// TIA Portal project "Connect_Winform" (V15)

(* hardware
DEVICE "S7-1200 station_1"  S7-1200 Station
   slot 0: "Rack_0"  S7-1200 Rack  Rack  V1.0
   slot 1: "PLC_1"  CPU 1214C DC/DC/Rly  6ES7 214-1HG40-0XB0  V4.2
   slot 2: "DI 16/DQ 16x24VDC_1"  SM 1223 DI16/DQ16 x 24VDC  6ES7 223-1BL30-0XB0  V1.0
*)

// ===== PLC "PLC_1"  CPU 1214C DC/DC/Rly =====

VAR_GLOBAL   // PLC tag table "Input"
   "Man" AT %I0.0 : Bool;
   "Silo1" AT %I0.1 : Bool;
   "Silo2" AT %I0.2 : Bool;
   "Silo3" AT %I0.3 : Bool;
   "Silo4" AT %I0.4 : Bool;
   "Silo5" AT %I0.5 : Bool;
   "Silo6" AT %I0.6 : Bool;
   "Silo7" AT %I0.7 : Bool;
   "Silo8" AT %I8.0 : Bool;
   "Silo9" AT %I8.1 : Bool;
   "Silo10" AT %I8.2 : Bool;
   "Silo11" AT %I8.3 : Bool;
   "Silo12" AT %I8.4 : Bool;
   "Silo13" AT %I8.5 : Bool;
   "Silo14" AT %I8.6 : Bool;
   "Silo15" AT %I8.7 : Bool;
   "Auto" AT %I9.0 : Bool;
   "InSilo" AT %I9.1 : Bool;
   "Mo Can" AT %I9.2 : Bool;
   "Dong Can" AT %I9.3 : Bool;
END_VAR

VAR_GLOBAL   // PLC tag table "Output"
   "Dang Can" AT %Q0.0 : Bool;
   "Silo_1" AT %Q0.1 : Bool;
   "Silo_2" AT %Q0.2 : Bool;
   "Silo_3" AT %Q0.3 : Bool;
   "Silo_4" AT %Q0.4 : Bool;
   "Silo_5" AT %Q0.5 : Bool;
   "Silo_6" AT %Q9.1 : Bool;
   "Silo_7" AT %Q9.2 : Bool;
   "Silo_8" AT %Q8.0 : Bool;
   "Silo_9" AT %Q8.1 : Bool;
   "Silo_10" AT %Q8.2 : Bool;
   "Silo_11" AT %Q8.3 : Bool;
   "Silo_12" AT %Q8.4 : Bool;
   "Silo_13" AT %Q8.5 : Bool;
   "Silo_14" AT %Q8.6 : Bool;
   "Silo_15" AT %Q8.7 : Bool;
   "Ngung Can" AT %Q9.0 : Bool;
   "Silo_16" AT %Q9.3 : Bool;
END_VAR

VAR_GLOBAL   // PLC tag table "Bien_Trung_Gian"
   "Bang_Tay" AT %M0.0 : Bool;
   "Sl1" AT %M0.1 : Bool;
   "Sl2" AT %M0.2 : Bool;
   "Sl3" AT %M0.3 : Bool;
   "Sl4" AT %M0.4 : Bool;
   "Sl5" AT %M0.5 : Bool;
   "Sl6" AT %M0.6 : Bool;
   "Sl7" AT %M0.7 : Bool;
   "Sl8" AT %M1.0 : Bool;
   "Sl9" AT %M1.1 : Bool;
   "Sl10" AT %M1.2 : Bool;
   "Sl11" AT %M1.3 : Bool;
   "Sl12" AT %M1.4 : Bool;
   "Sl13" AT %M1.5 : Bool;
   "Sl14" AT %M1.6 : Bool;
   "Sl15" AT %M1.7 : Bool;
   "Tu_Dong" AT %M2.0 : Bool;
   "Cho_Phep_Can1" AT %M2.1 : Bool;
   "Cho_Xa_Can" AT %M2.2 : Bool;
   "Sl16" AT %M2.3 : Bool;
   "Cho_Phep_Can2" AT %M2.4 : Bool;
   "Cho_Phep_Can3" AT %M2.5 : Bool;
END_VAR

DATA_BLOCK "DB_Winform"   // DB1
{ S7_Optimized_Access := 'FALSE' }
VERSION : 0.1
   VAR
      sn : Bool;
      Den2 : Bool;
      Den3 : Bool;
      Den4 : Bool;
      Den5 : Bool;
      Den6 : Bool;
      Den7 : Bool;
      Den8 : Bool;
      Den9 : Bool;
      Den10 : Bool;
      Den11 : Bool;
      Den12 : Bool;
      Den13 : Bool;
      Den14 : Bool;
      Den15 : Bool;
      Den16 : Bool;
      Den_CPC1 : Bool;
      Den_CPC2 : Bool;
      Den_CPC3 : Bool;
      end : Byte;
   END_VAR
BEGIN
END_DATA_BLOCK

DATA_BLOCK "FB1_Silo1"   // DB2
{ S7_Optimized_Access := 'TRUE' }
VERSION : 0.1
// stored: InstanceOfName FB1
"FB1"
BEGIN
END_DATA_BLOCK

DATA_BLOCK "FB1_Silo2"   // DB3
{ S7_Optimized_Access := 'TRUE' }
VERSION : 0.1
// stored: InstanceOfName FB1
"FB1"
BEGIN
END_DATA_BLOCK

DATA_BLOCK "FB1_Silo3"   // DB4
{ S7_Optimized_Access := 'TRUE' }
VERSION : 0.1
// stored: InstanceOfName FB1
"FB1"
BEGIN
END_DATA_BLOCK

DATA_BLOCK "FB1_Silo4"   // DB5
{ S7_Optimized_Access := 'TRUE' }
VERSION : 0.1
// stored: InstanceOfName FB1
"FB1"
BEGIN
END_DATA_BLOCK

DATA_BLOCK "FB1_Silo5"   // DB6
{ S7_Optimized_Access := 'TRUE' }
VERSION : 0.1
// stored: InstanceOfName FB1
"FB1"
BEGIN
END_DATA_BLOCK

DATA_BLOCK "FB1_Silo6"   // DB7
{ S7_Optimized_Access := 'TRUE' }
VERSION : 0.1
// stored: InstanceOfName FB1
"FB1"
BEGIN
END_DATA_BLOCK

DATA_BLOCK "FB1_Silo7"   // DB8
{ S7_Optimized_Access := 'TRUE' }
VERSION : 0.1
// stored: InstanceOfName FB1
"FB1"
BEGIN
END_DATA_BLOCK

DATA_BLOCK "FB1_Silo8"   // DB9
{ S7_Optimized_Access := 'TRUE' }
VERSION : 0.1
// stored: InstanceOfName FB1
"FB1"
BEGIN
END_DATA_BLOCK

DATA_BLOCK "FB1_Silo9"   // DB10
{ S7_Optimized_Access := 'TRUE' }
VERSION : 0.1
// stored: InstanceOfName FB1
"FB1"
BEGIN
END_DATA_BLOCK

DATA_BLOCK "FB1_Silo10"   // DB11
{ S7_Optimized_Access := 'TRUE' }
VERSION : 0.1
// stored: InstanceOfName FB1
"FB1"
BEGIN
END_DATA_BLOCK

DATA_BLOCK "FB1_Silo11"   // DB12
{ S7_Optimized_Access := 'TRUE' }
VERSION : 0.1
// stored: InstanceOfName FB1
"FB1"
BEGIN
END_DATA_BLOCK

DATA_BLOCK "FB1_Silo12"   // DB13
{ S7_Optimized_Access := 'TRUE' }
VERSION : 0.1
// stored: InstanceOfName FB1
"FB1"
BEGIN
END_DATA_BLOCK

DATA_BLOCK "FB1_Silo13"   // DB14
{ S7_Optimized_Access := 'TRUE' }
VERSION : 0.1
// stored: InstanceOfName FB1
"FB1"
BEGIN
END_DATA_BLOCK

DATA_BLOCK "FB1_Silo14"   // DB15
{ S7_Optimized_Access := 'TRUE' }
VERSION : 0.1
// stored: InstanceOfName FB1
"FB1"
BEGIN
END_DATA_BLOCK

DATA_BLOCK "FB1_Silo15"   // DB16
{ S7_Optimized_Access := 'TRUE' }
VERSION : 0.1
// stored: InstanceOfName FB1
"FB1"
BEGIN
END_DATA_BLOCK

DATA_BLOCK "FB1_Silo16"   // DB17
{ S7_Optimized_Access := 'TRUE' }
VERSION : 0.1
// stored: InstanceOfName FB1
"FB1"
BEGIN
END_DATA_BLOCK

FUNCTION_BLOCK "FB1"   // FB1, LAD
{ S7_Optimized_Access := 'TRUE' }
VERSION : 0.1
   VAR_INPUT
      Silo : Bool;
      "Silo+1" : Bool;
      "Silo+2" : Bool;
      "Silo+3" : Bool;
      "Silo+4" : Bool;
      "Silo+5" : Bool;
      "Silo+6" : Bool;
      "Silo+7" : Bool;
      "Silo+8" : Bool;
      "Silo+9" : Bool;
      "Silo+10" : Bool;
      "Silo+11" : Bool;
      "Silo+12" : Bool;
      "Silo+13" : Bool;
      "Silo+14" : Bool;
      "Silo+15" : Bool;
      In_Silo : Bool;
      Cho_Phep_Can : Bool;
      Nhan_Giu : Bool;
   END_VAR
   VAR_OUTPUT
      Silo_On : Bool;
   END_VAR
BEGIN

REGION Network 1
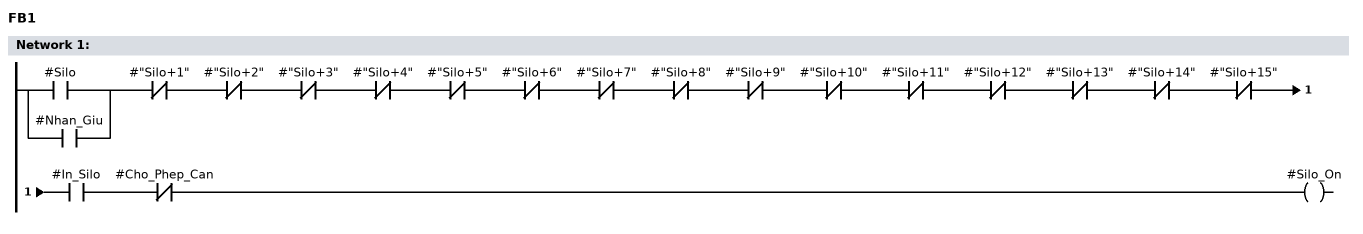
   RUNG wire#powerrail
      Contact( #Silo )
      wire#w1
      I_Contact( #"Silo+1" )
      I_Contact( #"Silo+2" )
      I_Contact( #"Silo+3" )
      I_Contact( #"Silo+4" )
      I_Contact( #"Silo+5" )
      I_Contact( #"Silo+6" )
      I_Contact( #"Silo+7" )
      I_Contact( #"Silo+8" )
      I_Contact( #"Silo+9" )
      I_Contact( #"Silo+10" )
      I_Contact( #"Silo+11" )
      I_Contact( #"Silo+12" )
      I_Contact( #"Silo+13" )
      I_Contact( #"Silo+14" )
      I_Contact( #"Silo+15" )
      Contact( #In_Silo )
      I_Contact( #Cho_Phep_Can )
      Coil( #Silo_On )
   END_RUNG
   RUNG wire#powerrail
      Contact( #Nhan_Giu )
   END_RUNG wire#w1
   // the same network as SCL:
   #Silo_On := (#Silo OR #Nhan_Giu) AND NOT #"Silo+1" AND NOT #"Silo+2" AND NOT #"Silo+3" AND NOT #"Silo+4" AND NOT #"Silo+5" AND NOT #"Silo+6" AND NOT #"Silo+7" AND NOT #"Silo+8" AND NOT #"Silo+9" AND NOT #"Silo+10" AND NOT #"Silo+11" AND NOT #"Silo+12" AND NOT #"Silo+13" AND NOT #"Silo+14" AND NOT #"Silo+15" AND #In_Silo AND NOT #Cho_Phep_Can;
END_REGION
END_FUNCTION_BLOCK

ORGANIZATION_BLOCK "Can"   // OB1, LAD, ProgramCycle
TITLE = "Main Program Sweep (Cycle)"
{ S7_Optimized_Access := 'TRUE' }
VERSION : 0.1
   VAR_INPUT
      Initial_Call : Bool;   // Initial call of this OB
      Remanence : Bool;   // =True, if remanent data are available
   END_VAR
BEGIN

REGION Network 1
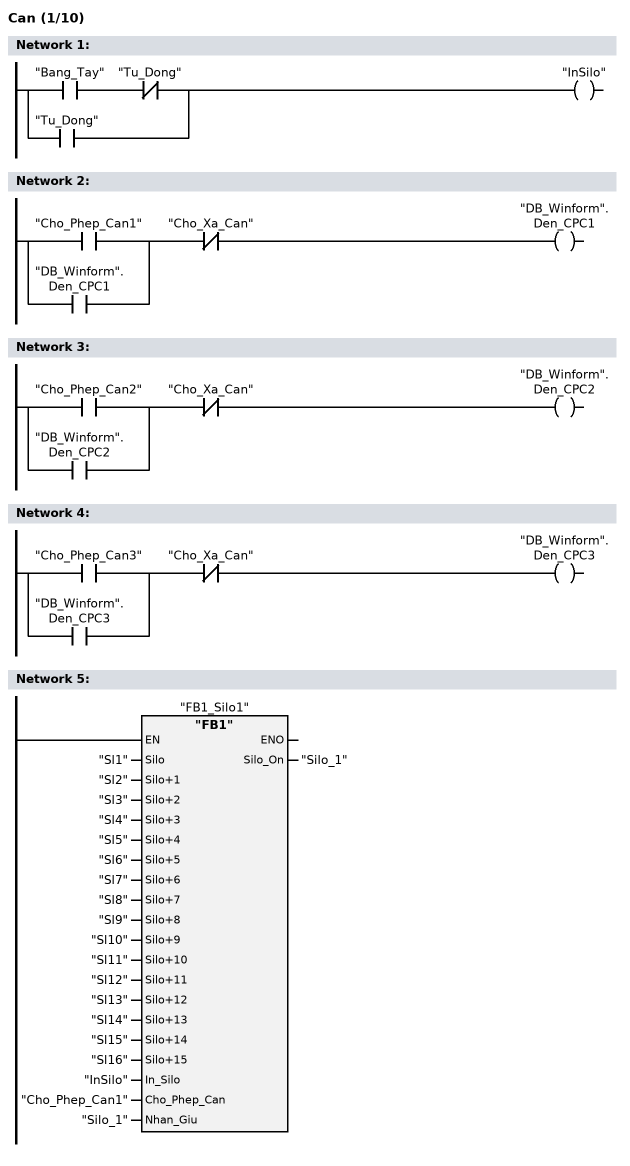
   RUNG wire#powerrail
      Contact( "Bang_Tay" )
      I_Contact( "Tu_Dong" )
      wire#w1
      Coil( "InSilo" )
   END_RUNG
   RUNG wire#powerrail
      Contact( "Tu_Dong" )
   END_RUNG wire#w1
   // the same network as SCL:
   "InSilo" := ("Bang_Tay" AND NOT "Tu_Dong") OR "Tu_Dong";
END_REGION

REGION Network 2
   RUNG wire#powerrail
      Contact( "Cho_Phep_Can1" )
      wire#w1
      I_Contact( "Cho_Xa_Can" )
      Coil( "DB_Winform".Den_CPC1 )
   END_RUNG
   RUNG wire#powerrail
      Contact( "DB_Winform".Den_CPC1 )
   END_RUNG wire#w1
   // the same network as SCL:
   "DB_Winform".Den_CPC1 := ("Cho_Phep_Can1" OR "DB_Winform".Den_CPC1) AND NOT "Cho_Xa_Can";
END_REGION

REGION Network 3
   RUNG wire#powerrail
      Contact( "Cho_Phep_Can2" )
      wire#w1
      I_Contact( "Cho_Xa_Can" )
      Coil( "DB_Winform".Den_CPC2 )
   END_RUNG
   RUNG wire#powerrail
      Contact( "DB_Winform".Den_CPC2 )
   END_RUNG wire#w1
   // the same network as SCL:
   "DB_Winform".Den_CPC2 := ("Cho_Phep_Can2" OR "DB_Winform".Den_CPC2) AND NOT "Cho_Xa_Can";
END_REGION

REGION Network 4
   RUNG wire#powerrail
      Contact( "Cho_Phep_Can3" )
      wire#w1
      I_Contact( "Cho_Xa_Can" )
      Coil( "DB_Winform".Den_CPC3 )
   END_RUNG
   RUNG wire#powerrail
      Contact( "DB_Winform".Den_CPC3 )
   END_RUNG wire#w1
   // the same network as SCL:
   "DB_Winform".Den_CPC3 := ("Cho_Phep_Can3" OR "DB_Winform".Den_CPC3) AND NOT "Cho_Xa_Can";
END_REGION

REGION Network 5
   RUNG wire#powerrail
      "FB1_Silo1"(Silo := "Sl1", "Silo+1" := "Sl2", "Silo+2" := "Sl3", "Silo+3" := "Sl4", "Silo+4" := "Sl5", "Silo+5" := "Sl6", "Silo+6" := "Sl7", "Silo+7" := "Sl8", "Silo+8" := "Sl9", "Silo+9" := "Sl10", "Silo+10" := "Sl11", "Silo+11" := "Sl12", "Silo+12" := "Sl13", "Silo+13" := "Sl14", "Silo+14" := "Sl15", "Silo+15" := "Sl16", In_Silo := "InSilo", Cho_Phep_Can := "Cho_Phep_Can1", Nhan_Giu := "Silo_1", Silo_On => "Silo_1")
   END_RUNG
   // the same network as SCL:
   "FB1_Silo1"(Silo := "Sl1",   // "FB1"
               "Silo+1" := "Sl2",
               "Silo+2" := "Sl3",
               "Silo+3" := "Sl4",
               "Silo+4" := "Sl5",
               "Silo+5" := "Sl6",
               "Silo+6" := "Sl7",
               "Silo+7" := "Sl8",
               "Silo+8" := "Sl9",
               "Silo+9" := "Sl10",
               "Silo+10" := "Sl11",
               "Silo+11" := "Sl12",
               "Silo+12" := "Sl13",
               "Silo+13" := "Sl14",
               "Silo+14" := "Sl15",
               "Silo+15" := "Sl16",
               In_Silo := "InSilo",
               Cho_Phep_Can := "Cho_Phep_Can1",
               Nhan_Giu := "Silo_1",
               Silo_On => "Silo_1");
END_REGION

REGION Network 6
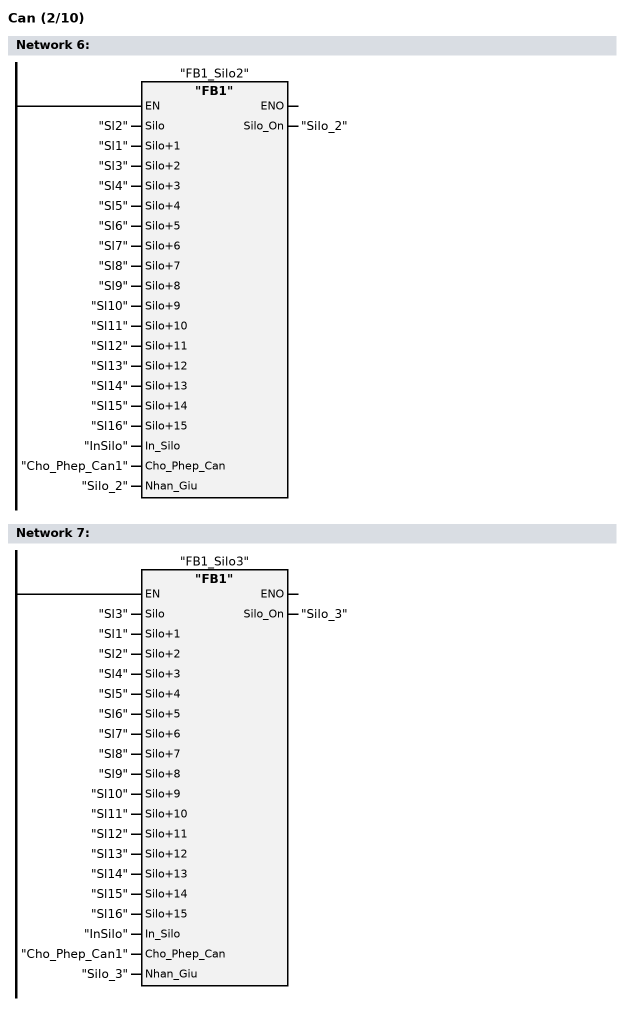
   RUNG wire#powerrail
      "FB1_Silo2"(Silo := "Sl2", "Silo+1" := "Sl1", "Silo+2" := "Sl3", "Silo+3" := "Sl4", "Silo+4" := "Sl5", "Silo+5" := "Sl6", "Silo+6" := "Sl7", "Silo+7" := "Sl8", "Silo+8" := "Sl9", "Silo+9" := "Sl10", "Silo+10" := "Sl11", "Silo+11" := "Sl12", "Silo+12" := "Sl13", "Silo+13" := "Sl14", "Silo+14" := "Sl15", "Silo+15" := "Sl16", In_Silo := "InSilo", Cho_Phep_Can := "Cho_Phep_Can1", Nhan_Giu := "Silo_2", Silo_On => "Silo_2")
   END_RUNG
   // the same network as SCL:
   "FB1_Silo2"(Silo := "Sl2",   // "FB1"
               "Silo+1" := "Sl1",
               "Silo+2" := "Sl3",
               "Silo+3" := "Sl4",
               "Silo+4" := "Sl5",
               "Silo+5" := "Sl6",
               "Silo+6" := "Sl7",
               "Silo+7" := "Sl8",
               "Silo+8" := "Sl9",
               "Silo+9" := "Sl10",
               "Silo+10" := "Sl11",
               "Silo+11" := "Sl12",
               "Silo+12" := "Sl13",
               "Silo+13" := "Sl14",
               "Silo+14" := "Sl15",
               "Silo+15" := "Sl16",
               In_Silo := "InSilo",
               Cho_Phep_Can := "Cho_Phep_Can1",
               Nhan_Giu := "Silo_2",
               Silo_On => "Silo_2");
END_REGION

REGION Network 7
   RUNG wire#powerrail
      "FB1_Silo3"(Silo := "Sl3", "Silo+1" := "Sl1", "Silo+2" := "Sl2", "Silo+3" := "Sl4", "Silo+4" := "Sl5", "Silo+5" := "Sl6", "Silo+6" := "Sl7", "Silo+7" := "Sl8", "Silo+8" := "Sl9", "Silo+9" := "Sl10", "Silo+10" := "Sl11", "Silo+11" := "Sl12", "Silo+12" := "Sl13", "Silo+13" := "Sl14", "Silo+14" := "Sl15", "Silo+15" := "Sl16", In_Silo := "InSilo", Cho_Phep_Can := "Cho_Phep_Can1", Nhan_Giu := "Silo_3", Silo_On => "Silo_3")
   END_RUNG
   // the same network as SCL:
   "FB1_Silo3"(Silo := "Sl3",   // "FB1"
               "Silo+1" := "Sl1",
               "Silo+2" := "Sl2",
               "Silo+3" := "Sl4",
               "Silo+4" := "Sl5",
               "Silo+5" := "Sl6",
               "Silo+6" := "Sl7",
               "Silo+7" := "Sl8",
               "Silo+8" := "Sl9",
               "Silo+9" := "Sl10",
               "Silo+10" := "Sl11",
               "Silo+11" := "Sl12",
               "Silo+12" := "Sl13",
               "Silo+13" := "Sl14",
               "Silo+14" := "Sl15",
               "Silo+15" := "Sl16",
               In_Silo := "InSilo",
               Cho_Phep_Can := "Cho_Phep_Can1",
               Nhan_Giu := "Silo_3",
               Silo_On => "Silo_3");
END_REGION

REGION Network 8
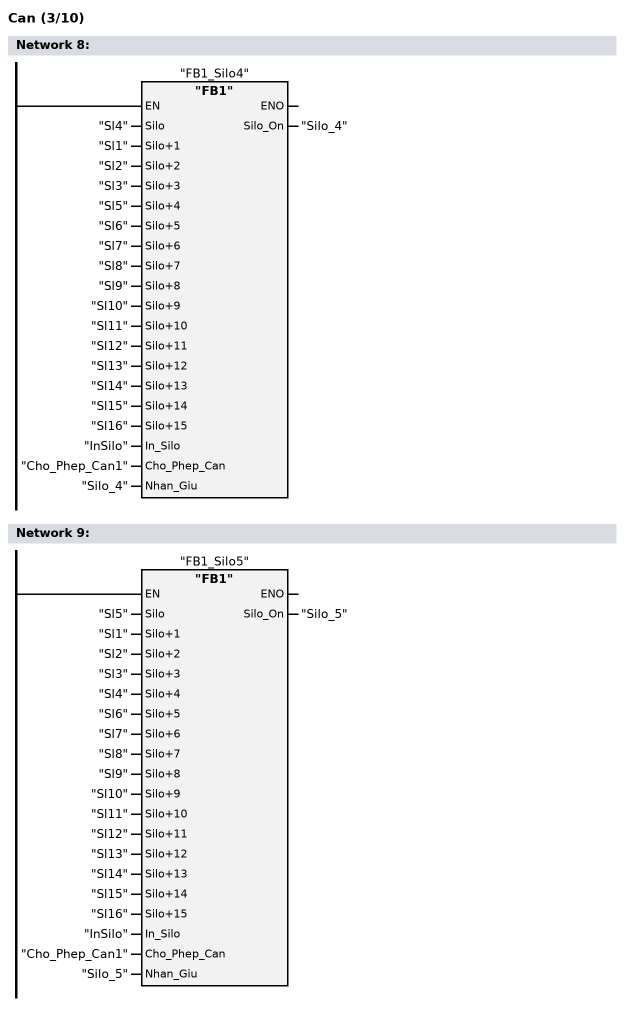
   RUNG wire#powerrail
      "FB1_Silo4"(Silo := "Sl4", "Silo+1" := "Sl1", "Silo+2" := "Sl2", "Silo+3" := "Sl3", "Silo+4" := "Sl5", "Silo+5" := "Sl6", "Silo+6" := "Sl7", "Silo+7" := "Sl8", "Silo+8" := "Sl9", "Silo+9" := "Sl10", "Silo+10" := "Sl11", "Silo+11" := "Sl12", "Silo+12" := "Sl13", "Silo+13" := "Sl14", "Silo+14" := "Sl15", "Silo+15" := "Sl16", In_Silo := "InSilo", Cho_Phep_Can := "Cho_Phep_Can1", Nhan_Giu := "Silo_4", Silo_On => "Silo_4")
   END_RUNG
   // the same network as SCL:
   "FB1_Silo4"(Silo := "Sl4",   // "FB1"
               "Silo+1" := "Sl1",
               "Silo+2" := "Sl2",
               "Silo+3" := "Sl3",
               "Silo+4" := "Sl5",
               "Silo+5" := "Sl6",
               "Silo+6" := "Sl7",
               "Silo+7" := "Sl8",
               "Silo+8" := "Sl9",
               "Silo+9" := "Sl10",
               "Silo+10" := "Sl11",
               "Silo+11" := "Sl12",
               "Silo+12" := "Sl13",
               "Silo+13" := "Sl14",
               "Silo+14" := "Sl15",
               "Silo+15" := "Sl16",
               In_Silo := "InSilo",
               Cho_Phep_Can := "Cho_Phep_Can1",
               Nhan_Giu := "Silo_4",
               Silo_On => "Silo_4");
END_REGION

REGION Network 9
   RUNG wire#powerrail
      "FB1_Silo5"(Silo := "Sl5", "Silo+1" := "Sl1", "Silo+2" := "Sl2", "Silo+3" := "Sl3", "Silo+4" := "Sl4", "Silo+5" := "Sl6", "Silo+6" := "Sl7", "Silo+7" := "Sl8", "Silo+8" := "Sl9", "Silo+9" := "Sl10", "Silo+10" := "Sl11", "Silo+11" := "Sl12", "Silo+12" := "Sl13", "Silo+13" := "Sl14", "Silo+14" := "Sl15", "Silo+15" := "Sl16", In_Silo := "InSilo", Cho_Phep_Can := "Cho_Phep_Can1", Nhan_Giu := "Silo_5", Silo_On => "Silo_5")
   END_RUNG
   // the same network as SCL:
   "FB1_Silo5"(Silo := "Sl5",   // "FB1"
               "Silo+1" := "Sl1",
               "Silo+2" := "Sl2",
               "Silo+3" := "Sl3",
               "Silo+4" := "Sl4",
               "Silo+5" := "Sl6",
               "Silo+6" := "Sl7",
               "Silo+7" := "Sl8",
               "Silo+8" := "Sl9",
               "Silo+9" := "Sl10",
               "Silo+10" := "Sl11",
               "Silo+11" := "Sl12",
               "Silo+12" := "Sl13",
               "Silo+13" := "Sl14",
               "Silo+14" := "Sl15",
               "Silo+15" := "Sl16",
               In_Silo := "InSilo",
               Cho_Phep_Can := "Cho_Phep_Can1",
               Nhan_Giu := "Silo_5",
               Silo_On => "Silo_5");
END_REGION

REGION Network 10
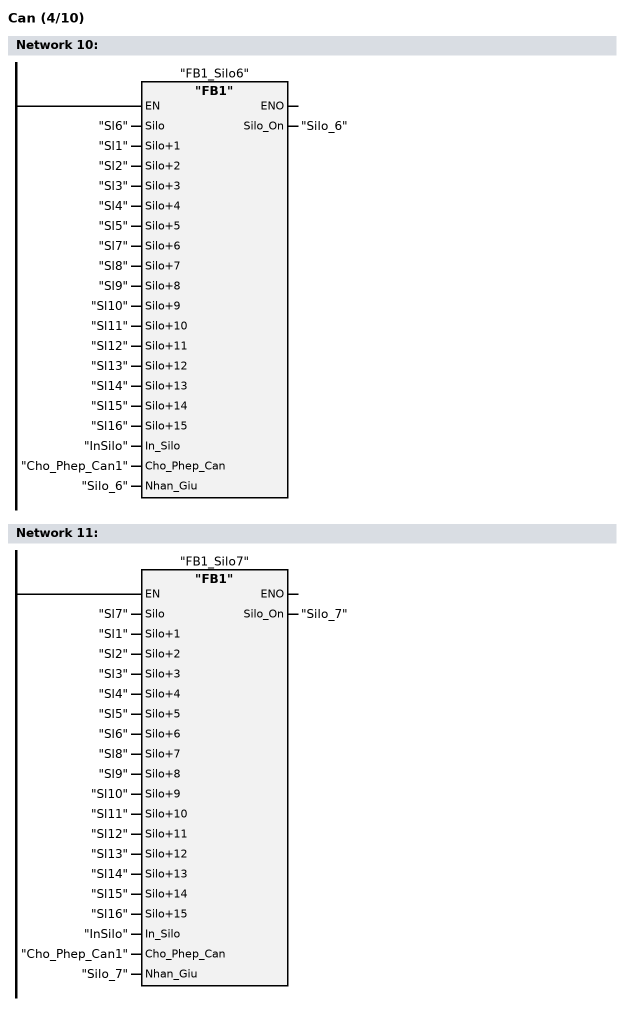
   RUNG wire#powerrail
      "FB1_Silo6"(Silo := "Sl6", "Silo+1" := "Sl1", "Silo+2" := "Sl2", "Silo+3" := "Sl3", "Silo+4" := "Sl4", "Silo+5" := "Sl5", "Silo+6" := "Sl7", "Silo+7" := "Sl8", "Silo+8" := "Sl9", "Silo+9" := "Sl10", "Silo+10" := "Sl11", "Silo+11" := "Sl12", "Silo+12" := "Sl13", "Silo+13" := "Sl14", "Silo+14" := "Sl15", "Silo+15" := "Sl16", In_Silo := "InSilo", Cho_Phep_Can := "Cho_Phep_Can1", Nhan_Giu := "Silo_6", Silo_On => "Silo_6")
   END_RUNG
   // the same network as SCL:
   "FB1_Silo6"(Silo := "Sl6",   // "FB1"
               "Silo+1" := "Sl1",
               "Silo+2" := "Sl2",
               "Silo+3" := "Sl3",
               "Silo+4" := "Sl4",
               "Silo+5" := "Sl5",
               "Silo+6" := "Sl7",
               "Silo+7" := "Sl8",
               "Silo+8" := "Sl9",
               "Silo+9" := "Sl10",
               "Silo+10" := "Sl11",
               "Silo+11" := "Sl12",
               "Silo+12" := "Sl13",
               "Silo+13" := "Sl14",
               "Silo+14" := "Sl15",
               "Silo+15" := "Sl16",
               In_Silo := "InSilo",
               Cho_Phep_Can := "Cho_Phep_Can1",
               Nhan_Giu := "Silo_6",
               Silo_On => "Silo_6");
END_REGION

REGION Network 11
   RUNG wire#powerrail
      "FB1_Silo7"(Silo := "Sl7", "Silo+1" := "Sl1", "Silo+2" := "Sl2", "Silo+3" := "Sl3", "Silo+4" := "Sl4", "Silo+5" := "Sl5", "Silo+6" := "Sl6", "Silo+7" := "Sl8", "Silo+8" := "Sl9", "Silo+9" := "Sl10", "Silo+10" := "Sl11", "Silo+11" := "Sl12", "Silo+12" := "Sl13", "Silo+13" := "Sl14", "Silo+14" := "Sl15", "Silo+15" := "Sl16", In_Silo := "InSilo", Cho_Phep_Can := "Cho_Phep_Can1", Nhan_Giu := "Silo_7", Silo_On => "Silo_7")
   END_RUNG
   // the same network as SCL:
   "FB1_Silo7"(Silo := "Sl7",   // "FB1"
               "Silo+1" := "Sl1",
               "Silo+2" := "Sl2",
               "Silo+3" := "Sl3",
               "Silo+4" := "Sl4",
               "Silo+5" := "Sl5",
               "Silo+6" := "Sl6",
               "Silo+7" := "Sl8",
               "Silo+8" := "Sl9",
               "Silo+9" := "Sl10",
               "Silo+10" := "Sl11",
               "Silo+11" := "Sl12",
               "Silo+12" := "Sl13",
               "Silo+13" := "Sl14",
               "Silo+14" := "Sl15",
               "Silo+15" := "Sl16",
               In_Silo := "InSilo",
               Cho_Phep_Can := "Cho_Phep_Can1",
               Nhan_Giu := "Silo_7",
               Silo_On => "Silo_7");
END_REGION

REGION Network 12
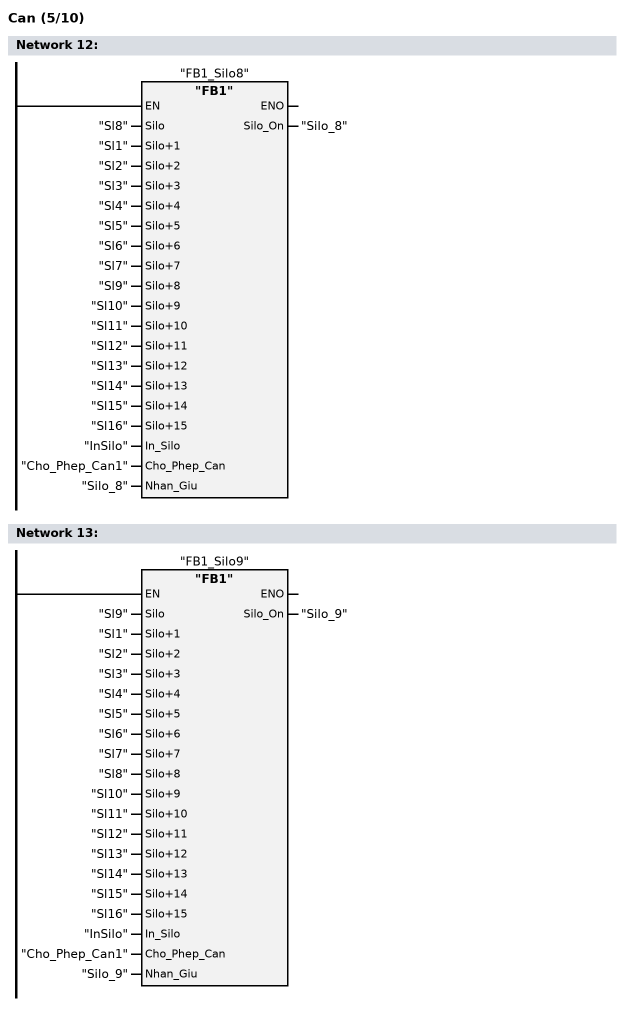
   RUNG wire#powerrail
      "FB1_Silo8"(Silo := "Sl8", "Silo+1" := "Sl1", "Silo+2" := "Sl2", "Silo+3" := "Sl3", "Silo+4" := "Sl4", "Silo+5" := "Sl5", "Silo+6" := "Sl6", "Silo+7" := "Sl7", "Silo+8" := "Sl9", "Silo+9" := "Sl10", "Silo+10" := "Sl11", "Silo+11" := "Sl12", "Silo+12" := "Sl13", "Silo+13" := "Sl14", "Silo+14" := "Sl15", "Silo+15" := "Sl16", In_Silo := "InSilo", Cho_Phep_Can := "Cho_Phep_Can1", Nhan_Giu := "Silo_8", Silo_On => "Silo_8")
   END_RUNG
   // the same network as SCL:
   "FB1_Silo8"(Silo := "Sl8",   // "FB1"
               "Silo+1" := "Sl1",
               "Silo+2" := "Sl2",
               "Silo+3" := "Sl3",
               "Silo+4" := "Sl4",
               "Silo+5" := "Sl5",
               "Silo+6" := "Sl6",
               "Silo+7" := "Sl7",
               "Silo+8" := "Sl9",
               "Silo+9" := "Sl10",
               "Silo+10" := "Sl11",
               "Silo+11" := "Sl12",
               "Silo+12" := "Sl13",
               "Silo+13" := "Sl14",
               "Silo+14" := "Sl15",
               "Silo+15" := "Sl16",
               In_Silo := "InSilo",
               Cho_Phep_Can := "Cho_Phep_Can1",
               Nhan_Giu := "Silo_8",
               Silo_On => "Silo_8");
END_REGION

REGION Network 13
   RUNG wire#powerrail
      "FB1_Silo9"(Silo := "Sl9", "Silo+1" := "Sl1", "Silo+2" := "Sl2", "Silo+3" := "Sl3", "Silo+4" := "Sl4", "Silo+5" := "Sl5", "Silo+6" := "Sl6", "Silo+7" := "Sl7", "Silo+8" := "Sl8", "Silo+9" := "Sl10", "Silo+10" := "Sl11", "Silo+11" := "Sl12", "Silo+12" := "Sl13", "Silo+13" := "Sl14", "Silo+14" := "Sl15", "Silo+15" := "Sl16", In_Silo := "InSilo", Cho_Phep_Can := "Cho_Phep_Can1", Nhan_Giu := "Silo_9", Silo_On => "Silo_9")
   END_RUNG
   // the same network as SCL:
   "FB1_Silo9"(Silo := "Sl9",   // "FB1"
               "Silo+1" := "Sl1",
               "Silo+2" := "Sl2",
               "Silo+3" := "Sl3",
               "Silo+4" := "Sl4",
               "Silo+5" := "Sl5",
               "Silo+6" := "Sl6",
               "Silo+7" := "Sl7",
               "Silo+8" := "Sl8",
               "Silo+9" := "Sl10",
               "Silo+10" := "Sl11",
               "Silo+11" := "Sl12",
               "Silo+12" := "Sl13",
               "Silo+13" := "Sl14",
               "Silo+14" := "Sl15",
               "Silo+15" := "Sl16",
               In_Silo := "InSilo",
               Cho_Phep_Can := "Cho_Phep_Can1",
               Nhan_Giu := "Silo_9",
               Silo_On => "Silo_9");
END_REGION

REGION Network 14
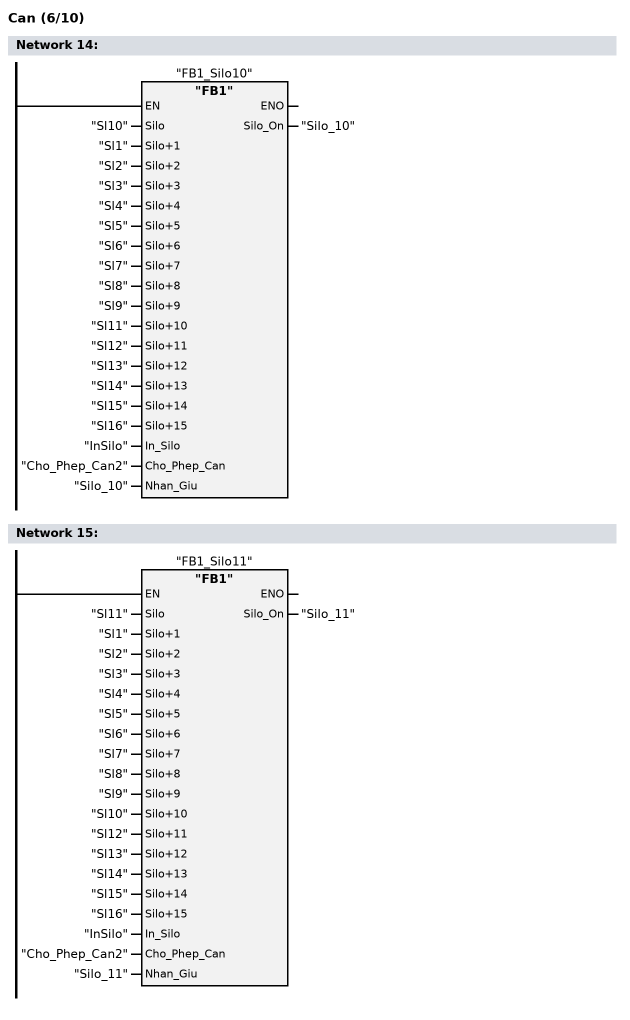
   RUNG wire#powerrail
      "FB1_Silo10"(Silo := "Sl10", "Silo+1" := "Sl1", "Silo+2" := "Sl2", "Silo+3" := "Sl3", "Silo+4" := "Sl4", "Silo+5" := "Sl5", "Silo+6" := "Sl6", "Silo+7" := "Sl7", "Silo+8" := "Sl8", "Silo+9" := "Sl9", "Silo+10" := "Sl11", "Silo+11" := "Sl12", "Silo+12" := "Sl13", "Silo+13" := "Sl14", "Silo+14" := "Sl15", "Silo+15" := "Sl16", In_Silo := "InSilo", Cho_Phep_Can := "Cho_Phep_Can2", Nhan_Giu := "Silo_10", Silo_On => "Silo_10")
   END_RUNG
   // the same network as SCL:
   "FB1_Silo10"(Silo := "Sl10",   // "FB1"
                "Silo+1" := "Sl1",
                "Silo+2" := "Sl2",
                "Silo+3" := "Sl3",
                "Silo+4" := "Sl4",
                "Silo+5" := "Sl5",
                "Silo+6" := "Sl6",
                "Silo+7" := "Sl7",
                "Silo+8" := "Sl8",
                "Silo+9" := "Sl9",
                "Silo+10" := "Sl11",
                "Silo+11" := "Sl12",
                "Silo+12" := "Sl13",
                "Silo+13" := "Sl14",
                "Silo+14" := "Sl15",
                "Silo+15" := "Sl16",
                In_Silo := "InSilo",
                Cho_Phep_Can := "Cho_Phep_Can2",
                Nhan_Giu := "Silo_10",
                Silo_On => "Silo_10");
END_REGION

REGION Network 15
   RUNG wire#powerrail
      "FB1_Silo11"(Silo := "Sl11", "Silo+1" := "Sl1", "Silo+2" := "Sl2", "Silo+3" := "Sl3", "Silo+4" := "Sl4", "Silo+5" := "Sl5", "Silo+6" := "Sl6", "Silo+7" := "Sl7", "Silo+8" := "Sl8", "Silo+9" := "Sl9", "Silo+10" := "Sl10", "Silo+11" := "Sl12", "Silo+12" := "Sl13", "Silo+13" := "Sl14", "Silo+14" := "Sl15", "Silo+15" := "Sl16", In_Silo := "InSilo", Cho_Phep_Can := "Cho_Phep_Can2", Nhan_Giu := "Silo_11", Silo_On => "Silo_11")
   END_RUNG
   // the same network as SCL:
   "FB1_Silo11"(Silo := "Sl11",   // "FB1"
                "Silo+1" := "Sl1",
                "Silo+2" := "Sl2",
                "Silo+3" := "Sl3",
                "Silo+4" := "Sl4",
                "Silo+5" := "Sl5",
                "Silo+6" := "Sl6",
                "Silo+7" := "Sl7",
                "Silo+8" := "Sl8",
                "Silo+9" := "Sl9",
                "Silo+10" := "Sl10",
                "Silo+11" := "Sl12",
                "Silo+12" := "Sl13",
                "Silo+13" := "Sl14",
                "Silo+14" := "Sl15",
                "Silo+15" := "Sl16",
                In_Silo := "InSilo",
                Cho_Phep_Can := "Cho_Phep_Can2",
                Nhan_Giu := "Silo_11",
                Silo_On => "Silo_11");
END_REGION

REGION Network 16
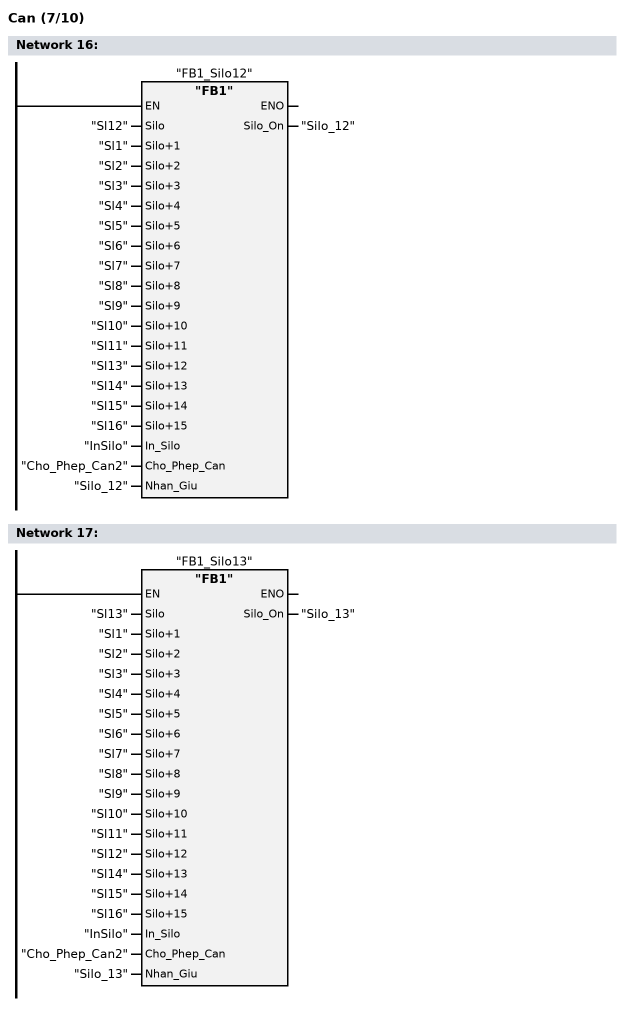
   RUNG wire#powerrail
      "FB1_Silo12"(Silo := "Sl12", "Silo+1" := "Sl1", "Silo+2" := "Sl2", "Silo+3" := "Sl3", "Silo+4" := "Sl4", "Silo+5" := "Sl5", "Silo+6" := "Sl6", "Silo+7" := "Sl7", "Silo+8" := "Sl8", "Silo+9" := "Sl9", "Silo+10" := "Sl10", "Silo+11" := "Sl11", "Silo+12" := "Sl13", "Silo+13" := "Sl14", "Silo+14" := "Sl15", "Silo+15" := "Sl16", In_Silo := "InSilo", Cho_Phep_Can := "Cho_Phep_Can2", Nhan_Giu := "Silo_12", Silo_On => "Silo_12")
   END_RUNG
   // the same network as SCL:
   "FB1_Silo12"(Silo := "Sl12",   // "FB1"
                "Silo+1" := "Sl1",
                "Silo+2" := "Sl2",
                "Silo+3" := "Sl3",
                "Silo+4" := "Sl4",
                "Silo+5" := "Sl5",
                "Silo+6" := "Sl6",
                "Silo+7" := "Sl7",
                "Silo+8" := "Sl8",
                "Silo+9" := "Sl9",
                "Silo+10" := "Sl10",
                "Silo+11" := "Sl11",
                "Silo+12" := "Sl13",
                "Silo+13" := "Sl14",
                "Silo+14" := "Sl15",
                "Silo+15" := "Sl16",
                In_Silo := "InSilo",
                Cho_Phep_Can := "Cho_Phep_Can2",
                Nhan_Giu := "Silo_12",
                Silo_On => "Silo_12");
END_REGION

REGION Network 17
   RUNG wire#powerrail
      "FB1_Silo13"(Silo := "Sl13", "Silo+1" := "Sl1", "Silo+2" := "Sl2", "Silo+3" := "Sl3", "Silo+4" := "Sl4", "Silo+5" := "Sl5", "Silo+6" := "Sl6", "Silo+7" := "Sl7", "Silo+8" := "Sl8", "Silo+9" := "Sl9", "Silo+10" := "Sl10", "Silo+11" := "Sl11", "Silo+12" := "Sl12", "Silo+13" := "Sl14", "Silo+14" := "Sl15", "Silo+15" := "Sl16", In_Silo := "InSilo", Cho_Phep_Can := "Cho_Phep_Can2", Nhan_Giu := "Silo_13", Silo_On => "Silo_13")
   END_RUNG
   // the same network as SCL:
   "FB1_Silo13"(Silo := "Sl13",   // "FB1"
                "Silo+1" := "Sl1",
                "Silo+2" := "Sl2",
                "Silo+3" := "Sl3",
                "Silo+4" := "Sl4",
                "Silo+5" := "Sl5",
                "Silo+6" := "Sl6",
                "Silo+7" := "Sl7",
                "Silo+8" := "Sl8",
                "Silo+9" := "Sl9",
                "Silo+10" := "Sl10",
                "Silo+11" := "Sl11",
                "Silo+12" := "Sl12",
                "Silo+13" := "Sl14",
                "Silo+14" := "Sl15",
                "Silo+15" := "Sl16",
                In_Silo := "InSilo",
                Cho_Phep_Can := "Cho_Phep_Can2",
                Nhan_Giu := "Silo_13",
                Silo_On => "Silo_13");
END_REGION

REGION Network 18
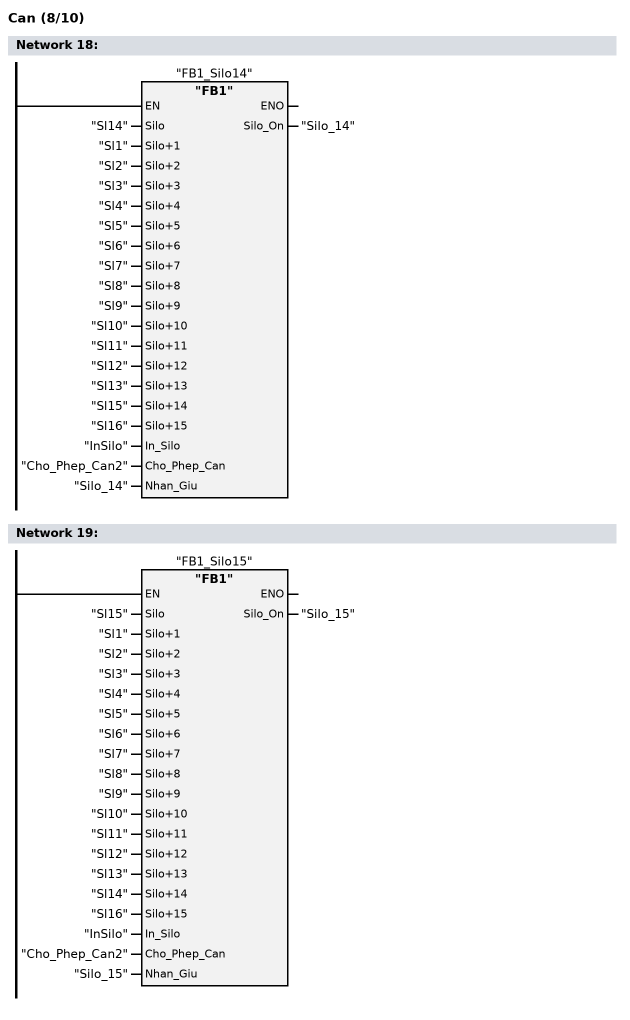
   RUNG wire#powerrail
      "FB1_Silo14"(Silo := "Sl14", "Silo+1" := "Sl1", "Silo+2" := "Sl2", "Silo+3" := "Sl3", "Silo+4" := "Sl4", "Silo+5" := "Sl5", "Silo+6" := "Sl6", "Silo+7" := "Sl7", "Silo+8" := "Sl8", "Silo+9" := "Sl9", "Silo+10" := "Sl10", "Silo+11" := "Sl11", "Silo+12" := "Sl12", "Silo+13" := "Sl13", "Silo+14" := "Sl15", "Silo+15" := "Sl16", In_Silo := "InSilo", Cho_Phep_Can := "Cho_Phep_Can2", Nhan_Giu := "Silo_14", Silo_On => "Silo_14")
   END_RUNG
   // the same network as SCL:
   "FB1_Silo14"(Silo := "Sl14",   // "FB1"
                "Silo+1" := "Sl1",
                "Silo+2" := "Sl2",
                "Silo+3" := "Sl3",
                "Silo+4" := "Sl4",
                "Silo+5" := "Sl5",
                "Silo+6" := "Sl6",
                "Silo+7" := "Sl7",
                "Silo+8" := "Sl8",
                "Silo+9" := "Sl9",
                "Silo+10" := "Sl10",
                "Silo+11" := "Sl11",
                "Silo+12" := "Sl12",
                "Silo+13" := "Sl13",
                "Silo+14" := "Sl15",
                "Silo+15" := "Sl16",
                In_Silo := "InSilo",
                Cho_Phep_Can := "Cho_Phep_Can2",
                Nhan_Giu := "Silo_14",
                Silo_On => "Silo_14");
END_REGION

REGION Network 19
   RUNG wire#powerrail
      "FB1_Silo15"(Silo := "Sl15", "Silo+1" := "Sl1", "Silo+2" := "Sl2", "Silo+3" := "Sl3", "Silo+4" := "Sl4", "Silo+5" := "Sl5", "Silo+6" := "Sl6", "Silo+7" := "Sl7", "Silo+8" := "Sl8", "Silo+9" := "Sl9", "Silo+10" := "Sl10", "Silo+11" := "Sl11", "Silo+12" := "Sl12", "Silo+13" := "Sl13", "Silo+14" := "Sl14", "Silo+15" := "Sl16", In_Silo := "InSilo", Cho_Phep_Can := "Cho_Phep_Can2", Nhan_Giu := "Silo_15", Silo_On => "Silo_15")
   END_RUNG
   // the same network as SCL:
   "FB1_Silo15"(Silo := "Sl15",   // "FB1"
                "Silo+1" := "Sl1",
                "Silo+2" := "Sl2",
                "Silo+3" := "Sl3",
                "Silo+4" := "Sl4",
                "Silo+5" := "Sl5",
                "Silo+6" := "Sl6",
                "Silo+7" := "Sl7",
                "Silo+8" := "Sl8",
                "Silo+9" := "Sl9",
                "Silo+10" := "Sl10",
                "Silo+11" := "Sl11",
                "Silo+12" := "Sl12",
                "Silo+13" := "Sl13",
                "Silo+14" := "Sl14",
                "Silo+15" := "Sl16",
                In_Silo := "InSilo",
                Cho_Phep_Can := "Cho_Phep_Can2",
                Nhan_Giu := "Silo_15",
                Silo_On => "Silo_15");
END_REGION

REGION Network 20
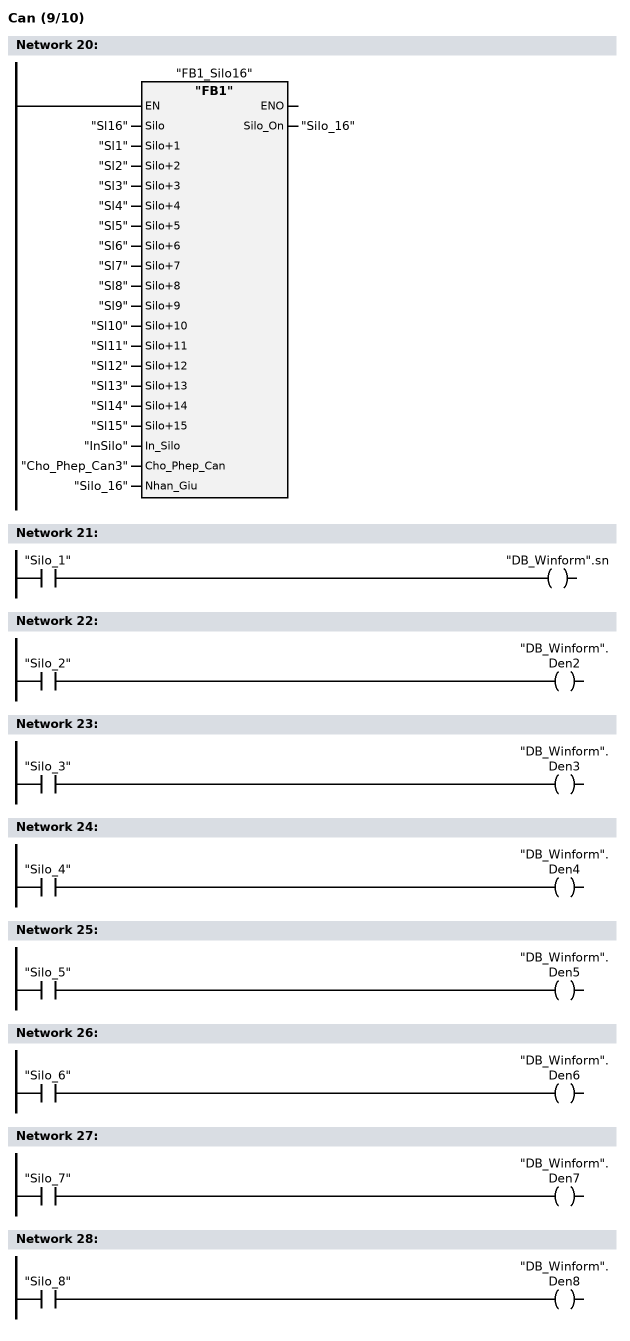
   RUNG wire#powerrail
      "FB1_Silo16"(Silo := "Sl16", "Silo+1" := "Sl1", "Silo+2" := "Sl2", "Silo+3" := "Sl3", "Silo+4" := "Sl4", "Silo+5" := "Sl5", "Silo+6" := "Sl6", "Silo+7" := "Sl7", "Silo+8" := "Sl8", "Silo+9" := "Sl9", "Silo+10" := "Sl10", "Silo+11" := "Sl11", "Silo+12" := "Sl12", "Silo+13" := "Sl13", "Silo+14" := "Sl14", "Silo+15" := "Sl15", In_Silo := "InSilo", Cho_Phep_Can := "Cho_Phep_Can3", Nhan_Giu := "Silo_16", Silo_On => "Silo_16")
   END_RUNG
   // the same network as SCL:
   "FB1_Silo16"(Silo := "Sl16",   // "FB1"
                "Silo+1" := "Sl1",
                "Silo+2" := "Sl2",
                "Silo+3" := "Sl3",
                "Silo+4" := "Sl4",
                "Silo+5" := "Sl5",
                "Silo+6" := "Sl6",
                "Silo+7" := "Sl7",
                "Silo+8" := "Sl8",
                "Silo+9" := "Sl9",
                "Silo+10" := "Sl10",
                "Silo+11" := "Sl11",
                "Silo+12" := "Sl12",
                "Silo+13" := "Sl13",
                "Silo+14" := "Sl14",
                "Silo+15" := "Sl15",
                In_Silo := "InSilo",
                Cho_Phep_Can := "Cho_Phep_Can3",
                Nhan_Giu := "Silo_16",
                Silo_On => "Silo_16");
END_REGION

REGION Network 21
   RUNG wire#powerrail
      Contact( "Silo_1" )
      Coil( "DB_Winform".sn )
   END_RUNG
   // the same network as SCL:
   "DB_Winform".sn := "Silo_1";
END_REGION

REGION Network 22
   RUNG wire#powerrail
      Contact( "Silo_2" )
      Coil( "DB_Winform".Den2 )
   END_RUNG
   // the same network as SCL:
   "DB_Winform".Den2 := "Silo_2";
END_REGION

REGION Network 23
   RUNG wire#powerrail
      Contact( "Silo_3" )
      Coil( "DB_Winform".Den3 )
   END_RUNG
   // the same network as SCL:
   "DB_Winform".Den3 := "Silo_3";
END_REGION

REGION Network 24
   RUNG wire#powerrail
      Contact( "Silo_4" )
      Coil( "DB_Winform".Den4 )
   END_RUNG
   // the same network as SCL:
   "DB_Winform".Den4 := "Silo_4";
END_REGION

REGION Network 25
   RUNG wire#powerrail
      Contact( "Silo_5" )
      Coil( "DB_Winform".Den5 )
   END_RUNG
   // the same network as SCL:
   "DB_Winform".Den5 := "Silo_5";
END_REGION

REGION Network 26
   RUNG wire#powerrail
      Contact( "Silo_6" )
      Coil( "DB_Winform".Den6 )
   END_RUNG
   // the same network as SCL:
   "DB_Winform".Den6 := "Silo_6";
END_REGION

REGION Network 27
   RUNG wire#powerrail
      Contact( "Silo_7" )
      Coil( "DB_Winform".Den7 )
   END_RUNG
   // the same network as SCL:
   "DB_Winform".Den7 := "Silo_7";
END_REGION

REGION Network 28
   RUNG wire#powerrail
      Contact( "Silo_8" )
      Coil( "DB_Winform".Den8 )
   END_RUNG
   // the same network as SCL:
   "DB_Winform".Den8 := "Silo_8";
END_REGION

REGION Network 29
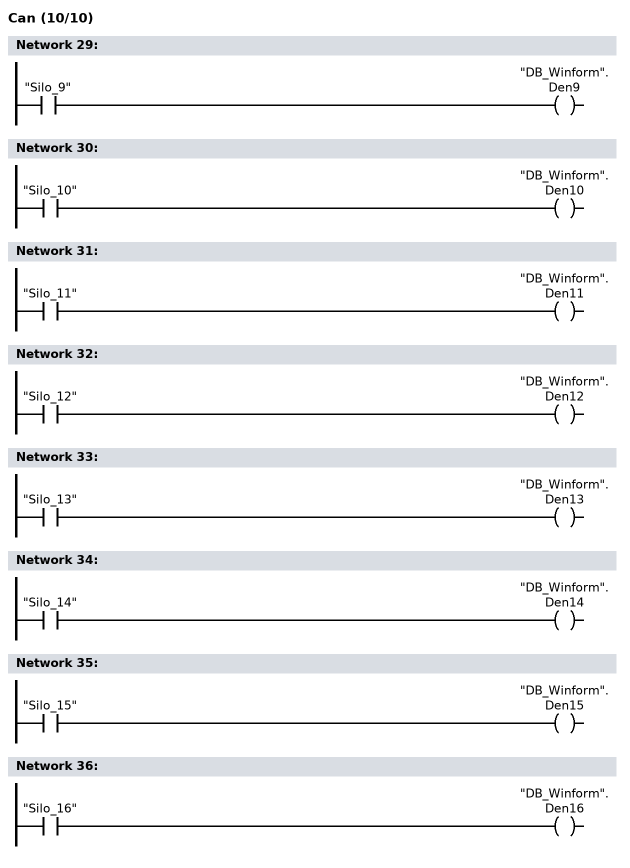
   RUNG wire#powerrail
      Contact( "Silo_9" )
      Coil( "DB_Winform".Den9 )
   END_RUNG
   // the same network as SCL:
   "DB_Winform".Den9 := "Silo_9";
END_REGION

REGION Network 30
   RUNG wire#powerrail
      Contact( "Silo_10" )
      Coil( "DB_Winform".Den10 )
   END_RUNG
   // the same network as SCL:
   "DB_Winform".Den10 := "Silo_10";
END_REGION

REGION Network 31
   RUNG wire#powerrail
      Contact( "Silo_11" )
      Coil( "DB_Winform".Den11 )
   END_RUNG
   // the same network as SCL:
   "DB_Winform".Den11 := "Silo_11";
END_REGION

REGION Network 32
   RUNG wire#powerrail
      Contact( "Silo_12" )
      Coil( "DB_Winform".Den12 )
   END_RUNG
   // the same network as SCL:
   "DB_Winform".Den12 := "Silo_12";
END_REGION

REGION Network 33
   RUNG wire#powerrail
      Contact( "Silo_13" )
      Coil( "DB_Winform".Den13 )
   END_RUNG
   // the same network as SCL:
   "DB_Winform".Den13 := "Silo_13";
END_REGION

REGION Network 34
   RUNG wire#powerrail
      Contact( "Silo_14" )
      Coil( "DB_Winform".Den14 )
   END_RUNG
   // the same network as SCL:
   "DB_Winform".Den14 := "Silo_14";
END_REGION

REGION Network 35
   RUNG wire#powerrail
      Contact( "Silo_15" )
      Coil( "DB_Winform".Den15 )
   END_RUNG
   // the same network as SCL:
   "DB_Winform".Den15 := "Silo_15";
END_REGION

REGION Network 36
   RUNG wire#powerrail
      Contact( "Silo_16" )
      Coil( "DB_Winform".Den16 )
   END_RUNG
   // the same network as SCL:
   "DB_Winform".Den16 := "Silo_16";
END_REGION
END_ORGANIZATION_BLOCK